// TIA Portal V17 export
// export: Created 2024-09-02T12:50:31.85908Z, ExportSetting WithDefaults, DisplayName Totally Integrated Automation Portal, DisplayVersion V17, DisplayName TIA Portal Openness, DisplayVersion V17, DisplayName TIA Portal Version Control Interface, DisplayVersion V17, DisplayName STEP 7 Professional, DisplayVersion V17, DisplayName STEP 7 Safety, DisplayVersion V17, DisplayName WinCC Professional, DisplayVersion V17
TYPE "UFM_UserRights"
TITLE = UFM_UserRights
// Describes the rights of the currently logges in user.
// stored: IsFailsafeCompliant false
   STRUCT
      RIGHT_ADMIN : Bool;   // User has administrative rights
      RIGHT_PRG_EDIT : Bool;   // User may edit programs
      RIGHT_STEP_EDIT : Bool;   // User may edit single program steps
      RIGHT_PRG_LOAD : Bool;   // User may load (select) a program
      RIGHT_MOVE : Bool;   // User may trigger axis movements
      RIGHT_CONFIG : Bool;   // User has configuration rights
   END_STRUCT;
END_TYPE
